# EPICS IOC start-up script: iocsh/EthercatMCslitAvoidCollSoftlimits.iocsh
dbLoadRecords("EthercatMCslitAvoidCollSoftlimits.template", "PREFIX=$(PREFIX), SLIT=$(SLIT), mXp=$(mXp), mXn=$(mXn) ")
